% RSLogix 500 project LINE 1 EAST_V2.00.RSS, saved by version 12.00.00.00 %
PROJECT "ML1400"    % processor: MicroLogix 1400; MAIN_PROG %

PROGRAM FILES
  LAD 2 "MAIN_PROG"  6 rungs
  LAD 3 "I/O"  9 rungs
  LAD 4 "WATER CTR"  10 rungs
  LAD 5 "PID"  4 rungs
  LAD 6 "ALARMS"  4 rungs
  LAD 7 "HMI"  25 rungs

DATA FILES
  O0 OUTPUT  10 elements
  I1 INPUT  26 elements
  S2 STATUS  66 elements
  B3 BINARY  32 elements
  T4 TIMER  16 elements
  C5 COUNTER  1 elements
  R6 CONTROL  1 elements
  N7 INTEGER  32 elements
  F8 FLOAT  32 elements
  B9 HMI BOOL  16 elements
  N10 HMI INT  16 elements
  PD11 PID  8 elements
  N12 PID INT  5 elements
  B13 FAULTS  1 elements
  N14 FAULTS  1 elements
  ST15 FAULTS  32 elements

LADDER 2 "MAIN_PROG"
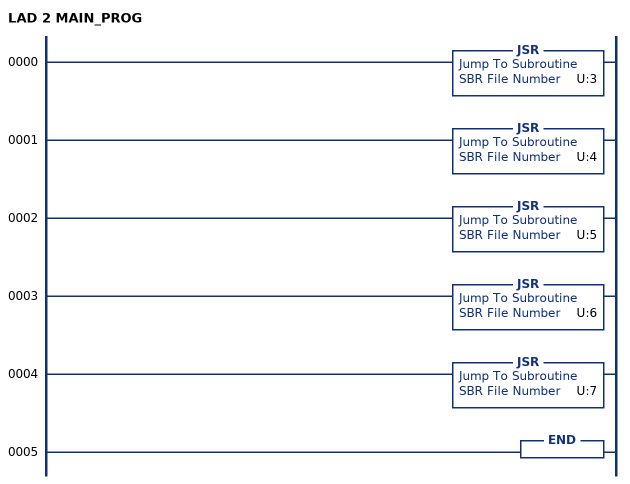
% Rung: 0 %
SOR JSR U:3 EOR
% Rung: 1 %
SOR JSR U:4 EOR
% Rung: 2 %
SOR JSR U:5 EOR
% Rung: 3 %
SOR JSR U:6 EOR
% Rung: 4 %
SOR JSR U:7 EOR
% Rung: 5 %
SOR END EOR

LADDER 3 "I/O"
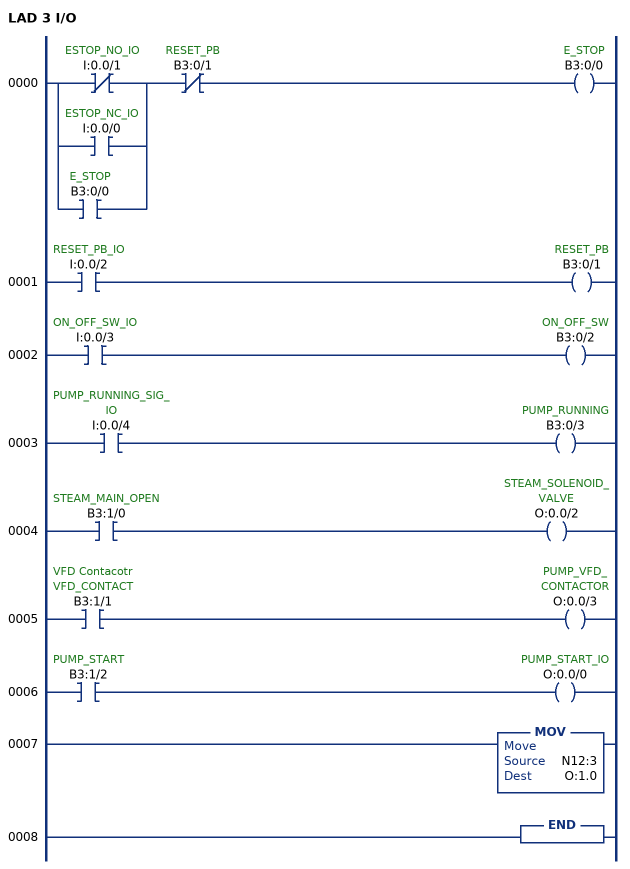
% Rung: 0 %
SOR BST XIO I:0.0/1 NXB XIC I:0.0/0 NXB XIC B3:0/0 BND XIO B3:0/1 OTE B3:0/0 EOR
%   I:0.0/1  ESTOP_NO_IO %
%   I:0.0/0  ESTOP_NC_IO %
%   B3:0/0  E_STOP %
%   B3:0/1  RESET_PB %
% Rung: 1 %
SOR XIC I:0.0/2 OTE B3:0/1 EOR
%   I:0.0/2  RESET_PB_IO %
%   B3:0/1  RESET_PB %
% Rung: 2 %
SOR XIC I:0.0/3 OTE B3:0/2 EOR
%   I:0.0/3  ON_OFF_SW_IO %
%   B3:0/2  ON_OFF_SW %
% Rung: 3 %
SOR XIC I:0.0/4 OTE B3:0/3 EOR
%   I:0.0/4  PUMP_RUNNING_SIG_IO %
%   B3:0/3  PUMP_RUNNING %
% Rung: 4 %
SOR XIC B3:1/0 OTE O:0.0/2 EOR
%   B3:1/0  STEAM_MAIN_OPEN %
%   O:0.0/2  STEAM_SOLENOID_VALVE %
% Rung: 5 %
SOR XIC B3:1/1 OTE O:0.0/3 EOR
%   B3:1/1  VFD_CONTACT  "VFD Contacotr" %
%   O:0.0/3  PUMP_VFD_CONTACTOR %
% Rung: 6 %
SOR XIC B3:1/2 OTE O:0.0/0 EOR
%   B3:1/2  PUMP_START %
%   O:0.0/0  PUMP_START_IO %
% Rung: 7 %
SOR MOV N12:3 O:1.0 EOR
%   N12:3  PID_OUT_SCALED %
% Rung: 8 %
SOR END EOR

LADDER 4 "WATER CTR"
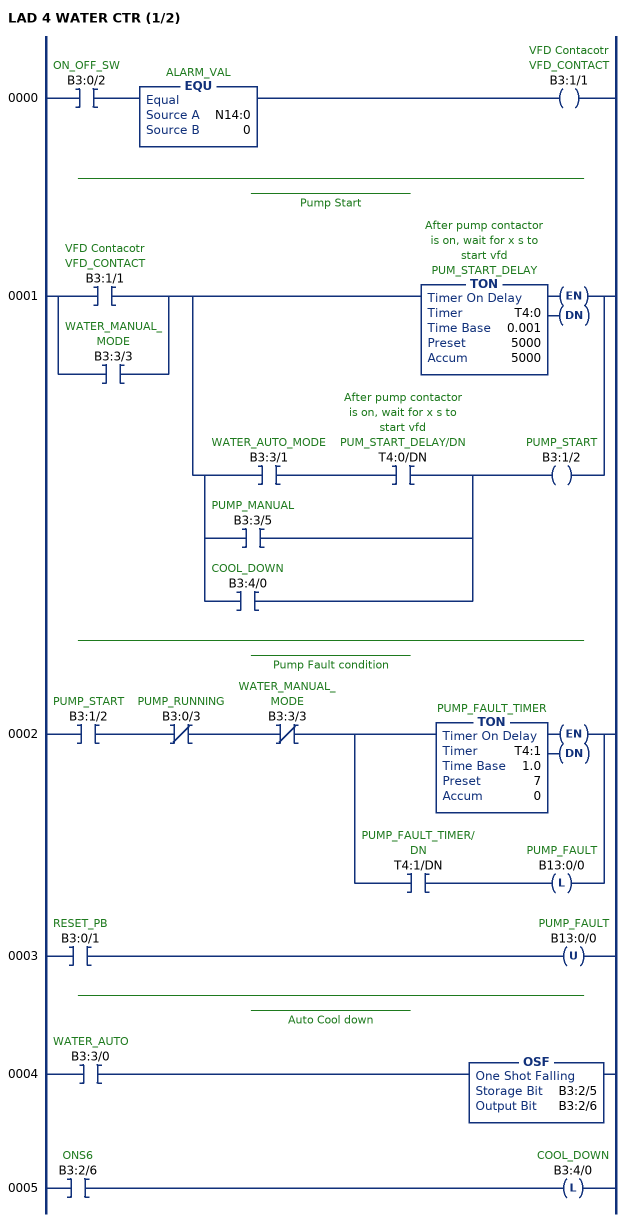
% Rung: 0 %
SOR XIC B3:0/2 EQU N14:0 0 OTE B3:1/1 EOR
%   B3:0/2  ON_OFF_SW %
%   N14:0  ALARM_VAL %
%   B3:1/1  VFD_CONTACT  "VFD Contacotr" %
% Rung: 1 %
% _________________________________________________________________________________________________________________________
% Pump Start %
SOR BST XIC B3:1/1 NXB XIC B3:3/3 BND BST TON T4:0 0.001 5000 5000 NXB BST XIC B3:3/1 XIC T4:0/DN NXB XIC B3:3/5 NXB XIC B3:4/0 BND OTE B3:1/2 BND EOR
%   B3:1/1  VFD_CONTACT  "VFD Contacotr" %
%   B3:3/3  WATER_MANUAL_MODE %
%   T4:0  PUM_START_DELAY  "After pump contactor is on, wait for x s to start vfd" %
%   B3:3/1  WATER_AUTO_MODE %
%   B3:3/5  PUMP_MANUAL %
%   B3:4/0  COOL_DOWN %
%   B3:1/2  PUMP_START %
% Rung: 2 %
% _________________________________________________________________________________________________________________________
% Pump Fault condition %
SOR XIC B3:1/2 XIO B3:0/3 XIO B3:3/3 BST TON T4:1 1.0 7 0 NXB XIC T4:1/DN OTL B13:0/0 BND EOR
%   B3:1/2  PUMP_START %
%   B3:0/3  PUMP_RUNNING %
%   B3:3/3  WATER_MANUAL_MODE %
%   T4:1  PUMP_FAULT_TIMER %
%   B13:0/0  PUMP_FAULT %
% Rung: 3 %
SOR XIC B3:0/1 OTU B13:0/0 EOR
%   B3:0/1  RESET_PB %
%   B13:0/0  PUMP_FAULT %
% Rung: 4 %
% _________________________________________________________________________________________________________________________
% Auto Cool down %
SOR XIC B3:3/0 OSF B3:2/5 B3:2/6 EOR
%   B3:3/0  WATER_AUTO %
%   B3:2/6  ONS6 %
% Rung: 5 %
SOR XIC B3:2/6 OTL B3:4/0 EOR
%   B3:2/6  ONS6 %
%   B3:4/0  COOL_DOWN %

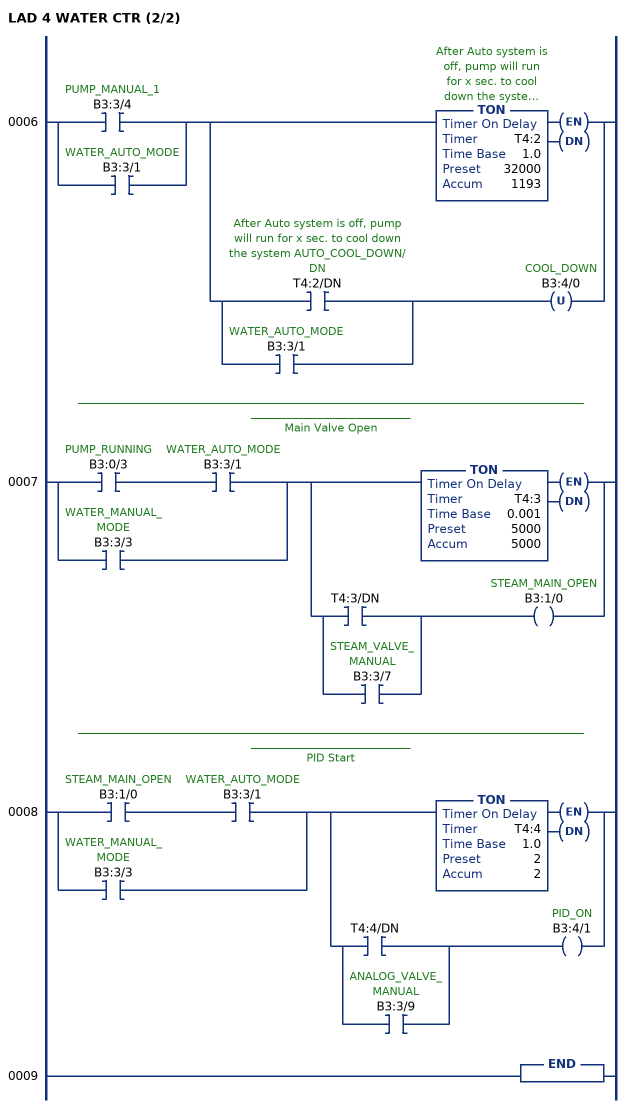
% Rung: 6 %
SOR BST XIC B3:3/4 NXB XIC B3:3/1 BND BST TON T4:2 1.0 32000 1193 NXB BST XIC T4:2/DN NXB XIC B3:3/1 BND OTU B3:4/0 BND EOR
%   B3:3/4  PUMP_MANUAL_1 %
%   B3:3/1  WATER_AUTO_MODE %
%   T4:2  AUTO_COOL_DOWN  "After Auto system is off, pump will run for x sec. to cool down the system" %
%   B3:4/0  COOL_DOWN %
% Rung: 7 %
% _________________________________________________________________________________________________________________________
% Main Valve Open %
SOR BST XIC B3:0/3 XIC B3:3/1 NXB XIC B3:3/3 BND BST TON T4:3 0.001 5000 5000 NXB BST XIC T4:3/DN NXB XIC B3:3/7 BND OTE B3:1/0 BND EOR
%   B3:0/3  PUMP_RUNNING %
%   B3:3/1  WATER_AUTO_MODE %
%   B3:3/3  WATER_MANUAL_MODE %
%   B3:3/7  STEAM_VALVE_MANUAL %
%   B3:1/0  STEAM_MAIN_OPEN %
% Rung: 8 %
% _________________________________________________________________________________________________________________________
% PID Start %
SOR BST XIC B3:1/0 XIC B3:3/1 NXB XIC B3:3/3 BND BST TON T4:4 1.0 2 2 NXB BST XIC T4:4/DN NXB XIC B3:3/9 BND OTE B3:4/1 BND EOR
%   B3:1/0  STEAM_MAIN_OPEN %
%   B3:3/1  WATER_AUTO_MODE %
%   B3:3/3  WATER_MANUAL_MODE %
%   B3:3/9  ANALOG_VALVE_MANUAL %
%   B3:4/1  PID_ON %
% Rung: 9 %
SOR END EOR

LADDER 5 "PID"
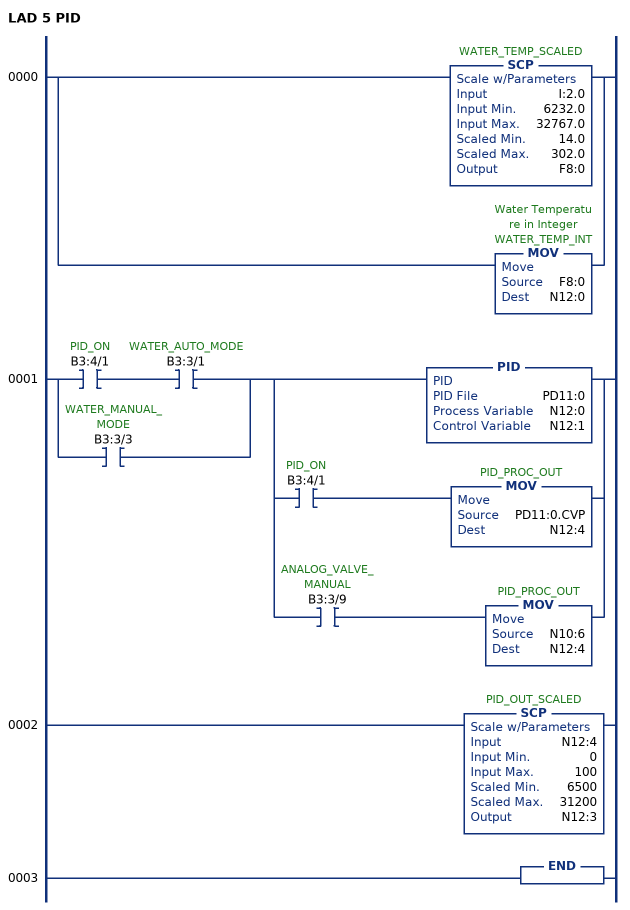
% Rung: 0 %
SOR BST SCP I:2.0 6232.0 32767.0 14.0 302.0 F8:0 NXB MOV F8:0 N12:0 BND EOR
%   I:2.0  WATER_TEMP_INPUT %
%   F8:0  WATER_TEMP_SCALED %
%   N12:0  WATER_TEMP_INT  "Water Temperature in Integer" %
% Rung: 1 %
SOR BST XIC B3:4/1 XIC B3:3/1 NXB XIC B3:3/3 BND BST PID PD11:0 N12:0 N12:1 NXB BST XIC B3:4/1 MOV PD11:0.CVP N12:4 NXB XIC B3:3/9 MOV N10:6 N12:4 BND BND EOR
%   B3:4/1  PID_ON %
%   B3:3/1  WATER_AUTO_MODE %
%   B3:3/3  WATER_MANUAL_MODE %
%   N12:0  WATER_TEMP_INT  "Water Temperature in Integer" %
%   N12:1  PID_OUT %
%   N12:4  PID_PROC_OUT %
%   B3:3/9  ANALOG_VALVE_MANUAL %
%   N10:6  HMI_PROP_VALVE_OPEN %
% Rung: 2 %
SOR SCP N12:4 0 100 6500 31200 N12:3 EOR
%   N12:4  PID_PROC_OUT %
%   N12:3  PID_OUT_SCALED %
% Rung: 3 %
SOR END EOR

LADDER 6 "ALARMS"
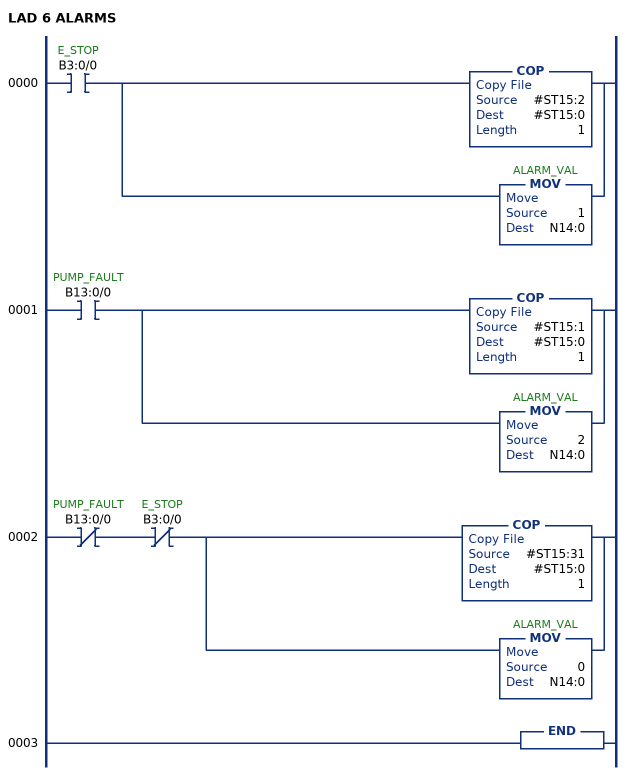
% Rung: 0 %
SOR XIC B3:0/0 BST COP #ST15:2 #ST15:0 1 NXB MOV 1 N14:0 BND EOR
%   B3:0/0  E_STOP %
%   N14:0  ALARM_VAL %
% Rung: 1 %
SOR XIC B13:0/0 BST COP #ST15:1 #ST15:0 1 NXB MOV 2 N14:0 BND EOR
%   B13:0/0  PUMP_FAULT %
%   N14:0  ALARM_VAL %
% Rung: 2 %
SOR XIO B13:0/0 XIO B3:0/0 BST COP #ST15:31 #ST15:0 1 NXB MOV 0 N14:0 BND EOR
%   B13:0/0  PUMP_FAULT %
%   B3:0/0  E_STOP %
%   N14:0  ALARM_VAL %
% Rung: 3 %
SOR END EOR

LADDER 7 "HMI"
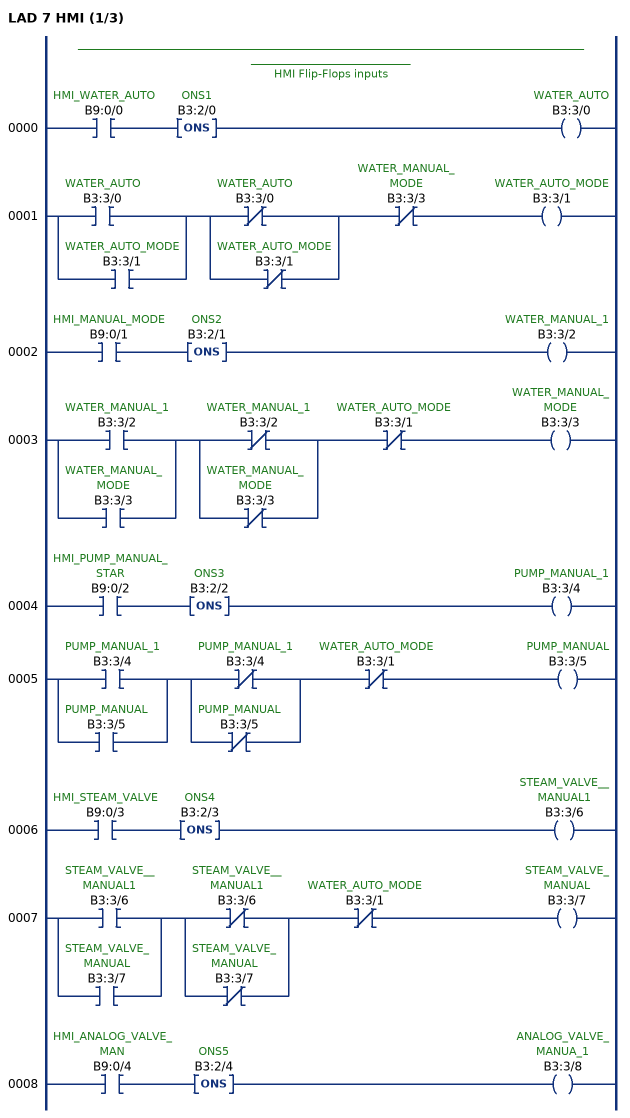
% Rung: 0 %
% _________________________________________________________________________________________________________________________
% HMI Flip-Flops inputs %
SOR XIC B9:0/0 ONS B3:2/0 OTE B3:3/0 EOR
%   B9:0/0  HMI_WATER_AUTO %
%   B3:2/0  ONS1 %
%   B3:3/0  WATER_AUTO %
% Rung: 1 %
SOR BST XIC B3:3/0 NXB XIC B3:3/1 BND BST XIO B3:3/0 NXB XIO B3:3/1 BND XIO B3:3/3 OTE B3:3/1 EOR
%   B3:3/0  WATER_AUTO %
%   B3:3/1  WATER_AUTO_MODE %
%   B3:3/3  WATER_MANUAL_MODE %
% Rung: 2 %
SOR XIC B9:0/1 ONS B3:2/1 OTE B3:3/2 EOR
%   B9:0/1  HMI_MANUAL_MODE %
%   B3:2/1  ONS2 %
%   B3:3/2  WATER_MANUAL_1 %
% Rung: 3 %
SOR BST XIC B3:3/2 NXB XIC B3:3/3 BND BST XIO B3:3/2 NXB XIO B3:3/3 BND XIO B3:3/1 OTE B3:3/3 EOR
%   B3:3/2  WATER_MANUAL_1 %
%   B3:3/3  WATER_MANUAL_MODE %
%   B3:3/1  WATER_AUTO_MODE %
% Rung: 4 %
SOR XIC B9:0/2 ONS B3:2/2 OTE B3:3/4 EOR
%   B9:0/2  HMI_PUMP_MANUAL_STAR %
%   B3:2/2  ONS3 %
%   B3:3/4  PUMP_MANUAL_1 %
% Rung: 5 %
SOR BST XIC B3:3/4 NXB XIC B3:3/5 BND BST XIO B3:3/4 NXB XIO B3:3/5 BND XIO B3:3/1 OTE B3:3/5 EOR
%   B3:3/4  PUMP_MANUAL_1 %
%   B3:3/5  PUMP_MANUAL %
%   B3:3/1  WATER_AUTO_MODE %
% Rung: 6 %
SOR XIC B9:0/3 ONS B3:2/3 OTE B3:3/6 EOR
%   B9:0/3  HMI_STEAM_VALVE %
%   B3:2/3  ONS4 %
%   B3:3/6  STEAM_VALVE__MANUAL1 %
% Rung: 7 %
SOR BST XIC B3:3/6 NXB XIC B3:3/7 BND BST XIO B3:3/6 NXB XIO B3:3/7 BND XIO B3:3/1 OTE B3:3/7 EOR
%   B3:3/6  STEAM_VALVE__MANUAL1 %
%   B3:3/7  STEAM_VALVE_MANUAL %
%   B3:3/1  WATER_AUTO_MODE %
% Rung: 8 %
SOR XIC B9:0/4 ONS B3:2/4 OTE B3:3/8 EOR
%   B9:0/4  HMI_ANALOG_VALVE_MAN %
%   B3:2/4  ONS5 %
%   B3:3/8  ANALOG_VALVE_MANUA_1 %

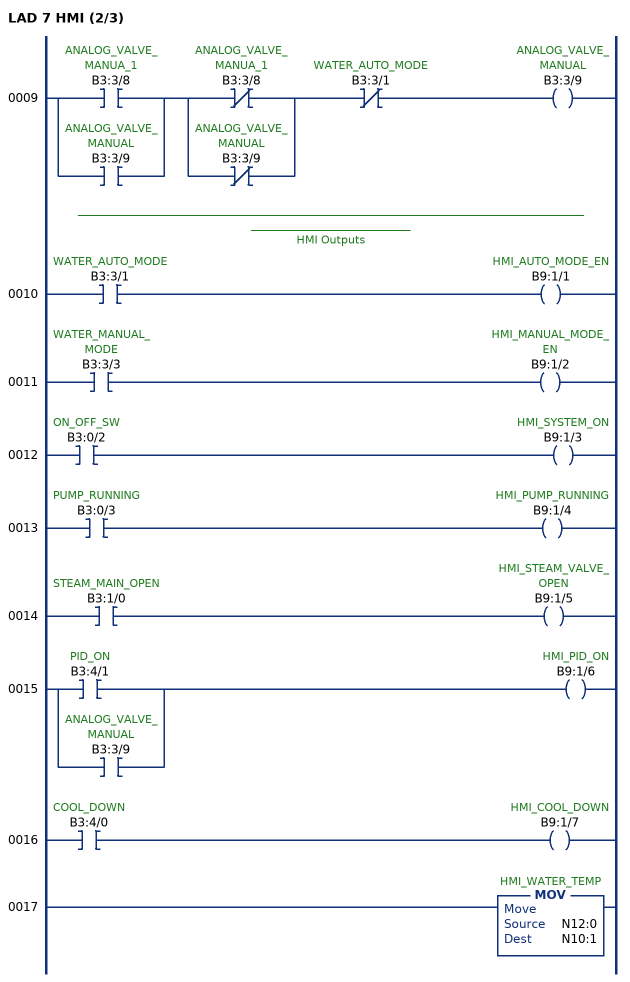
% Rung: 9 %
SOR BST XIC B3:3/8 NXB XIC B3:3/9 BND BST XIO B3:3/8 NXB XIO B3:3/9 BND XIO B3:3/1 OTE B3:3/9 EOR
%   B3:3/8  ANALOG_VALVE_MANUA_1 %
%   B3:3/9  ANALOG_VALVE_MANUAL %
%   B3:3/1  WATER_AUTO_MODE %
% Rung: 10 %
% _________________________________________________________________________________________________________________________
% HMI Outputs %
SOR XIC B3:3/1 OTE B9:1/1 EOR
%   B3:3/1  WATER_AUTO_MODE %
%   B9:1/1  HMI_AUTO_MODE_EN %
% Rung: 11 %
SOR XIC B3:3/3 OTE B9:1/2 EOR
%   B3:3/3  WATER_MANUAL_MODE %
%   B9:1/2  HMI_MANUAL_MODE_EN %
% Rung: 12 %
SOR XIC B3:0/2 OTE B9:1/3 EOR
%   B3:0/2  ON_OFF_SW %
%   B9:1/3  HMI_SYSTEM_ON %
% Rung: 13 %
SOR XIC B3:0/3 OTE B9:1/4 EOR
%   B3:0/3  PUMP_RUNNING %
%   B9:1/4  HMI_PUMP_RUNNING %
% Rung: 14 %
SOR XIC B3:1/0 OTE B9:1/5 EOR
%   B3:1/0  STEAM_MAIN_OPEN %
%   B9:1/5  HMI_STEAM_VALVE_OPEN %
% Rung: 15 %
SOR BST XIC B3:4/1 NXB XIC B3:3/9 BND OTE B9:1/6 EOR
%   B3:4/1  PID_ON %
%   B3:3/9  ANALOG_VALVE_MANUAL %
%   B9:1/6  HMI_PID_ON %
% Rung: 16 %
SOR XIC B3:4/0 OTE B9:1/7 EOR
%   B3:4/0  COOL_DOWN %
%   B9:1/7  HMI_COOL_DOWN %
% Rung: 17 %
SOR MOV N12:0 N10:1 EOR
%   N12:0  WATER_TEMP_INT  "Water Temperature in Integer" %
%   N10:1  HMI_WATER_TEMP %

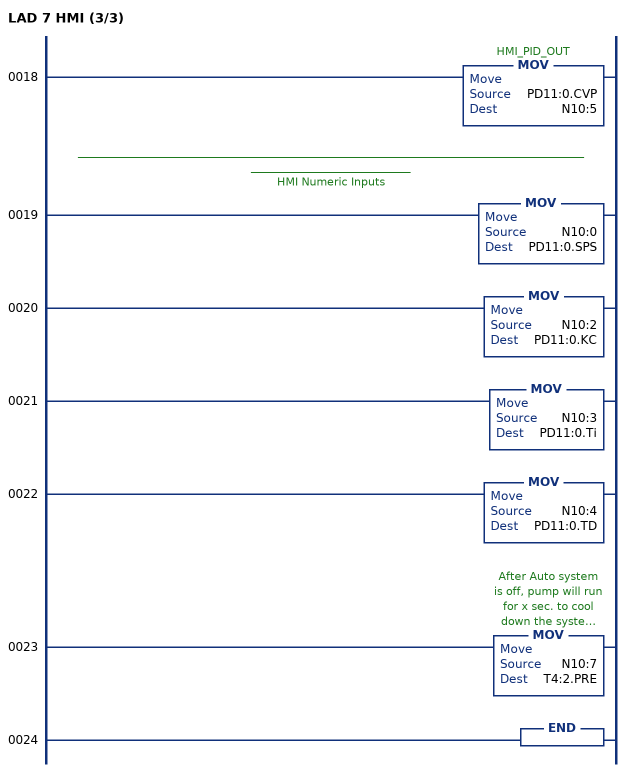
% Rung: 18 %
SOR MOV PD11:0.CVP N10:5 EOR
%   N10:5  HMI_PID_OUT %
% Rung: 19 %
% _________________________________________________________________________________________________________________________
% HMI Numeric Inputs %
SOR MOV N10:0 PD11:0.SPS EOR
%   N10:0  HMI_WATER_SETPOINT %
% Rung: 20 %
SOR MOV N10:2 PD11:0.KC EOR
%   N10:2  HMI_PID_KC %
% Rung: 21 %
SOR MOV N10:3 PD11:0.Ti EOR
%   N10:3  HMI_PID_TI %
% Rung: 22 %
SOR MOV N10:4 PD11:0.TD EOR
%   N10:4  HMI_PID_TD %
% Rung: 23 %
SOR MOV N10:7 T4:2.PRE EOR
%   N10:7  HMI_COOL_DOWN_TIME %
%   T4:2  AUTO_COOL_DOWN  "After Auto system is off, pump will run for x sec. to cool down the system" %
% Rung: 24 %
SOR END EOR

OTHER DOCUMENTED ADDRESSES
  B9:1/0  HMI_READY_TO_START
  F10:0  WATER_TEMP_SCACLED  "Water Temperature"
  F10:1  WATER_TEMP_FILTERED  "Water Temperature Filtered"
  N12:2  PID_OUT_X2
  N15:0  HMI_AUTO_COOL_TIME
  PD11:0.2  PID_WATER_SETPOINT

DATA TABLE (non-zero values as saved)
DATA B3
% B3:0 % 0X000C 0X0407 0X0000 0X0002 0X0002 0X0000 0X0000 0X0000 0X0000 0X0000
DATA T4
% .PRE .ACC %
% T4:0 % 5000 5000
% T4:1 % 7 0
% T4:2 % 32000 1193
% T4:3 % 5000 5000
% T4:4 % 2 2
DATA N7
% N7:0 % 77 757 50 0 0 0 0 0 0 0
DATA F8
% F8:0 % 100.5682 0 0 0 0
DATA B9
% B9:0 % 0X0000 0X007A 0X0000 0X0000 0X0000 0X0000 0X0000 0X0000 0X0000 0X0000
DATA N10
% N10:0 % 100 101 5800 29000 1 19 0 32000 0 0
DATA N12
% N12:0 % 100 3740 0 12181 23
DATA ST15
% ST15:1 % "Pump Faulted"
% ST15:2 % "E-Stop Pressed"
